// TIA Portal project "Flugnummer" (V20)

(* hardware
DEVICE "S7-1500/ET200MP-Station_1"  S7-1500 station
   slot 0: "Profilschiene_0"  Rack  6ES7 590-1***0-0AA0
   slot 1: "PLC_1"  CPU 1513-1 PN  6ES7 513-1AM03-0AB0  V4.0
      slot 3: "CPU-Display_1"  6ES7591-1AA00-0AA0
      slot 32768: "PROFINET-Schnittstelle_1"  X1
         slot 32769: "Port_1"  X1 P1
         slot 32770: "Port_2"  X1 P2
      slot 34817: "Virtual CP interface port_1"  Virtual CP interface port  Virtual CP interface port FW V4.0
   slot 2: "DI 16x24VDC BA_1"  DI 16x24VDC BA  6ES7 521-1BH10-0AA0  V1.1
   slot 3: "DQ 16x24VDC/0.5A ST_1"  DQ 16x24VDC/0.5A ST  6ES7 522-1BH00-0AB0  V2.0
   slot 4: "AI 8xU/I/R/RTD BA_1"  AI 8xU/I/R/RTD BA  6ES7 531-7QF00-0AB0  V1.0
   slot 5: "AQ 8xU/I HS_1"  AQ 8xU/I HS  6ES7 532-5HF00-0AB0  V2.2
   slot 6: "AI 8xU/I/R/RTD BA_2"  AI 8xU/I/R/RTD BA  6ES7 531-7QF00-0AB0  V1.0
   slot 7: "AQ 8xU/I HS_2"  AQ 8xU/I HS  6ES7 532-5HF00-0AB0  V2.2
*)

// ===== PLC "PLC_1"  CPU 1513-1 PN =====

VAR_GLOBAL   // PLC tag table "Standard-Variablentabelle"
   "PlcLabConnectIn01" AT %ID32760 : DWord;
   "PlcLabConnectIn02" AT %ID32764 : DWord;
   "PlcLabConnectOut01" AT %QD32760 : DWord;
   "PlcLabConnectOut02" AT %QD32764 : DWord;
   "Einschalter" AT %E0.0 : Bool;
   "Zurücksetzen" AT %E0.1 : Bool;
   "Leer" AT %M0.0 : Bool;
END_VAR

DATA_BLOCK "Datenbaustein_1"   // DB1
{ S7_Optimized_Access := 'TRUE' }
VERSION : 0.1
   VAR
      Eingabe : Struct
         Vorname : String := 'Maximilian';
         Nachname : String := 'Mustermann';
         Flugnummer : String := '123456789';
         Start : String := 'Hannover';
         Ziel : String := 'Paris';
      END_STRUCT;
      Ausgabe : Struct
         Buchungsnummer : String;
      END_STRUCT;
   END_VAR
BEGIN
END_DATA_BLOCK

ORGANIZATION_BLOCK "Main"   // OB1, FBD, ProgramCycle
TITLE = "Main Program Sweep (Cycle)"
{ S7_Optimized_Access := 'TRUE' }
VERSION : 0.1
   VAR_INPUT
      Initial_Call : Bool;   // Initial call of this OB
      Remanence : Bool;   // =True, if remanent data are available
   END_VAR
   VAR_TEMP
      VName : String;
      NName : String;
      SStadt : String;
      ZStadt : String;
   END_VAR
   VAR_TEMP   // added for the SCL form of the ladder/FBD networks
      _w1 : Bool;
   END_VAR
BEGIN

REGION Network 1
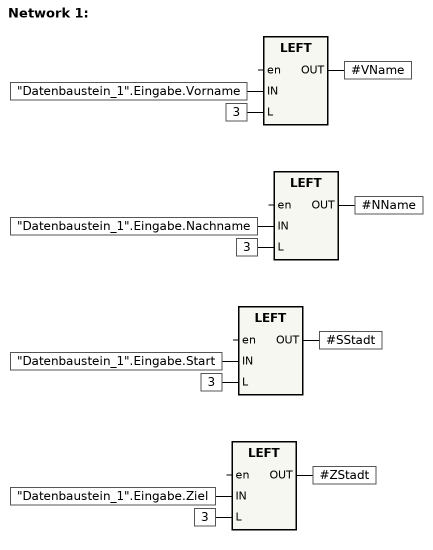
   #VName := LEFT(IN := "Datenbaustein_1".Eingabe.Vorname, L := 3);
   #NName := LEFT(IN := "Datenbaustein_1".Eingabe.Nachname, L := 3);
   #SStadt := LEFT(IN := "Datenbaustein_1".Eingabe.Start, L := 3);
   #ZStadt := LEFT(IN := "Datenbaustein_1".Eingabe.Ziel, L := 3);
END_REGION

REGION Network 2
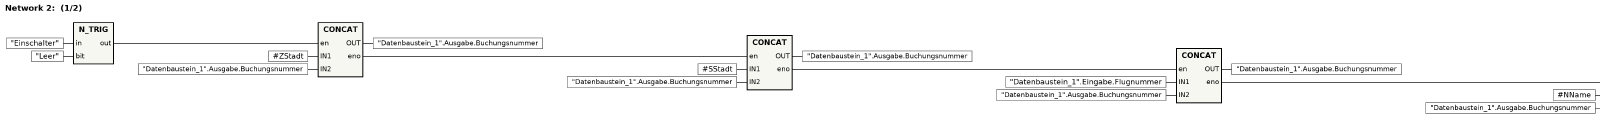
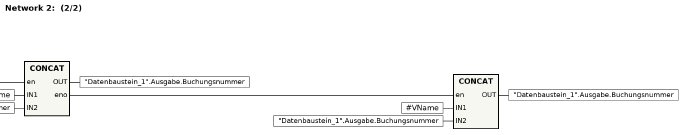
   #_w1 := NOT "Einschalter" AND "Leer";   // falling edge
   "Leer" := "Einschalter";
   IF #_w1 THEN
       "Datenbaustein_1".Ausgabe.Buchungsnummer := CONCAT(IN1 := #ZStadt,
                               IN2 := "Datenbaustein_1".Ausgabe.Buchungsnummer);
       "Datenbaustein_1".Ausgabe.Buchungsnummer := CONCAT(IN1 := #SStadt,
                               IN2 := "Datenbaustein_1".Ausgabe.Buchungsnummer);
       "Datenbaustein_1".Ausgabe.Buchungsnummer := CONCAT(IN1 := "Datenbaustein_1".Eingabe.Flugnummer,
                               IN2 := "Datenbaustein_1".Ausgabe.Buchungsnummer);
       "Datenbaustein_1".Ausgabe.Buchungsnummer := CONCAT(IN1 := #NName,
                               IN2 := "Datenbaustein_1".Ausgabe.Buchungsnummer);
       "Datenbaustein_1".Ausgabe.Buchungsnummer := CONCAT(IN1 := #VName,
                               IN2 := "Datenbaustein_1".Ausgabe.Buchungsnummer);
   END_IF;
END_REGION

REGION Network 3
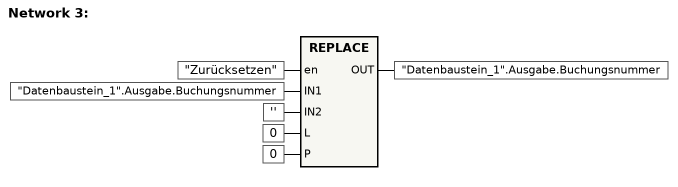
   IF "Zurücksetzen" THEN
       "Datenbaustein_1".Ausgabe.Buchungsnummer := REPLACE(IN1 := "Datenbaustein_1".Ausgabe.Buchungsnummer,
                               IN2 := '',
                               L := 0,
                               P := 0);
   END_IF;
END_REGION
END_ORGANIZATION_BLOCK